         (*********************************************)
         (* parameter 3.4.7 *)
         (*********************************************)
         (
            ParameterName_as8    := 'Output Value 43',
            ParameterType_u8     := 0,
            attr1_u              := 0,
            attr2_u              := 10000,
            attr3_u              := 50,
            UnitCode_au8         := 15,
            Multiplier_s16       := 1,
            Divisor_s16          := 1,
            NumberOfDigits_u16   := 0,
            AccesslevelCode_u8   := 129,
            attr4_u              := 0,
            EEPROMAddress_s      := (Page_u8 := 3, IntIndex_u8 := 158)
         ),

         (*********************************************)
         (* parameter 3.4.8 *)
         (*********************************************)
         (
            ParameterName_as8    := 'Output Value 44',
            ParameterType_u8     := 0,
            attr1_u              := 0,
            attr2_u              := 10000,
            attr3_u              := 50,
            UnitCode_au8         := 15,
            Multiplier_s16       := 1,
            Divisor_s16          := 1,
            NumberOfDigits_u16   := 0,
            AccesslevelCode_u8   := 129,
            attr4_u              := 0,
            EEPROMAddress_s      := (Page_u8 := 3, IntIndex_u8 := 159)
         )

      ),

      (*********************************************)
      (* parameter group 3.5 - up to 8 parameters can be defined here *)
      (*********************************************)
      (
         GroupName_as8   := 'Output Value 45-47',

         Param_as        := 

         (*********************************************)
         (* parameter 3.5.1 *)
         (*********************************************)
         (
            ParameterName_as8    := 'Output Value 45',
            ParameterType_u8     := 0,
            attr1_u              := 0,
            attr2_u              := 10000,
            attr3_u              := 50,
            UnitCode_au8         := 15,
            Multiplier_s16       := 1,
            Divisor_s16          := 1,
            NumberOfDigits_u16   := 0,
            AccesslevelCode_u8   := 129,
            attr4_u              := 0,
            EEPROMAddress_s      := (Page_u8 := 3, IntIndex_u8 := 160)
         ),

         (*********************************************)
         (* parameter 3.5.2 *)
         (*********************************************)
         (
            ParameterName_as8    := 'Output Value 46',
            ParameterType_u8     := 0,
            attr1_u              := 0,
            attr2_u              := 10000,
            attr3_u              := 50,
            UnitCode_au8         := 15,
            Multiplier_s16       := 1,
            Divisor_s16          := 1,
            NumberOfDigits_u16   := 0,
            AccesslevelCode_u8   := 129,
            attr4_u              := 0,
            EEPROMAddress_s      := (Page_u8 := 3, IntIndex_u8 := 161)
         ),

         (*********************************************)
         (* parameter 3.5.3 *)
         (*********************************************)
         (
            ParameterName_as8    := 'Output Value 47',
            ParameterType_u8     := 0,
            attr1_u              := 0,
            attr2_u              := 20000,
            attr3_u              := 50,
            UnitCode_au8         := 15,
            Multiplier_s16       := 1,
            Divisor_s16          := 1,
            NumberOfDigits_u16   := 0,
            AccesslevelCode_u8   := 129,
            attr4_u              := 0,
            EEPROMAddress_s      := (Page_u8 := 3, IntIndex_u8 := 162)
         ),

         (*********************************************)
         (* parameter 3.5.4 *)
         (*********************************************)
         (
         ),

         (*********************************************)
         (* parameter 3.5.5 *)
         (*********************************************)
         (
         ),

         (*********************************************)
         (* parameter 3.5.6 *)
         (*********************************************)
         (
         ),

         (*********************************************)
         (* parameter 3.5.7 *)
         (*********************************************)
         (
         ),

         (*********************************************)
         (* parameter 3.5.8 *)
         (*********************************************)
         (
         )

      ),

      (*********************************************)
      (* parameter group 3.6 - up to 8 parameters can be defined here *)
      (*********************************************)
      (
         GroupName_as8   := 'POH Configuration',

         Param_as        := 

         (*********************************************)
         (* parameter 3.6.1 *)
         (*********************************************)
         (
            ParameterName_as8    := 'POH Debounce',
            ParameterType_u8     := 0,
            attr1_u              := 50,
            attr2_u              := 250,
            attr3_u              := 10,
            UnitCode_au8         := 4,
            Multiplier_s16       := 1,
            Divisor_s16          := 1,
            NumberOfDigits_u16   := 0,
            AccesslevelCode_u8   := 179,
            attr4_u              := 100,
            EEPROMAddress_s      := (Page_u8 := 3, IntIndex_u8 := 168)
         ),

         (*********************************************)
         (* parameter 3.6.2 *)
         (*********************************************)
         (
         ),

         (*********************************************)
         (* parameter 3.6.3 *)
         (*********************************************)
         (
            ParameterName_as8    := 'POH Resistance Min',
            ParameterType_u8     := 0,
            attr1_u              := 0,
            attr2_u              := 3000,
            attr3_u              := 10,
            UnitCode_au8         := 18,
            Multiplier_s16       := 1,
            Divisor_s16          := 1,
            NumberOfDigits_u16   := 0,
            AccesslevelCode_u8   := 179,
            attr4_u              := 2,
            EEPROMAddress_s      := (Page_u8 := 3, IntIndex_u8 := 170)
         ),

         (*********************************************)
         (* parameter 3.6.4 *)
         (*********************************************)
         (
            ParameterName_as8    := 'POH Resistance Max',
            ParameterType_u8     := 0,
            attr1_u              := 0,
            attr2_u              := 3000,
            attr3_u              := 10,
            UnitCode_au8         := 18,
            Multiplier_s16       := 1,
            Divisor_s16          := 1,
            NumberOfDigits_u16   := 0,
            AccesslevelCode_u8   := 179,
            attr4_u              := 52,
            EEPROMAddress_s      := (Page_u8 := 3, IntIndex_u8 := 171)
         ),

         (*********************************************)
         (* parameter 3.6.5 *)
         (*********************************************)
         (
            ParameterName_as8    := 'POH Kp',
            ParameterType_u8     := 0,
            attr1_u              := 0,
            attr2_u              := 2000,
            attr3_u              := 50,
            UnitCode_au8         := 0,
            Multiplier_s16       := 1,
            Divisor_s16          := 1,
            NumberOfDigits_u16   := 0,
            AccesslevelCode_u8   := 179,
            attr4_u              := 250,
            EEPROMAddress_s      := (Page_u8 := 3, IntIndex_u8 := 172)
         ),

         (*********************************************)
         (* parameter 3.6.6 *)
         (*********************************************)
         (
            ParameterName_as8    := 'POH Ki',
            ParameterType_u8     := 0,
            attr1_u              := 0,
            attr2_u              := 500,
            attr3_u              := 50,
            UnitCode_au8         := 0,
            Multiplier_s16       := 1,
            Divisor_s16          := 1,
            NumberOfDigits_u16   := 0,
            AccesslevelCode_u8   := 179,
            attr4_u              := 250,
            EEPROMAddress_s      := (Page_u8 := 3, IntIndex_u8 := 173)
         ),

         (*********************************************)
         (* parameter 3.6.7 *)
         (*********************************************)
         (
         ),

         (*********************************************)
         (* parameter 3.6.8 *)
         (*********************************************)
         (
         )

      ),

      (*********************************************)
      (* parameter group 3.7 - up to 8 parameters can be defined here *)
      (*********************************************)
      (
         GroupName_as8   := 'POL Configuration',

         Param_as        := 

         (*********************************************)
         (* parameter 3.7.1 *)
         (*********************************************)
         (
            ParameterName_as8    := 'POL Debounce',
            ParameterType_u8     := 0,
            attr1_u              := 50,
            attr2_u              := 250,
            attr3_u              := 10,
            UnitCode_au8         := 4,
            Multiplier_s16       := 1,
            Divisor_s16          := 1,
            NumberOfDigits_u16   := 0,
            AccesslevelCode_u8   := 179,
            attr4_u              := 100,
            EEPROMAddress_s      := (Page_u8 := 3, IntIndex_u8 := 176)
         ),

         (*********************************************)
         (* parameter 3.7.2 *)
         (*********************************************)
         (
         ),

         (*********************************************)
         (* parameter 3.7.3 *)
         (*********************************************)
         (
            ParameterName_as8    := 'POL Resistance Min',
            ParameterType_u8     := 0,
            attr1_u              := 0,
            attr2_u              := 3000,
            attr3_u              := 10,
            UnitCode_au8         := 18,
            Multiplier_s16       := 1,
            Divisor_s16          := 1,
            NumberOfDigits_u16   := 0,
            AccesslevelCode_u8   := 179,
            attr4_u              := 2,
            EEPROMAddress_s      := (Page_u8 := 3, IntIndex_u8 := 178)
         ),

         (*********************************************)
         (* parameter 3.7.4 *)
         (*********************************************)
         (
            ParameterName_as8    := 'POL Resistance Max',
            ParameterType_u8     := 0,
            attr1_u              := 0,
            attr2_u              := 3000,
            attr3_u              := 10,
            UnitCode_au8         := 18,
            Multiplier_s16       := 1,
            Divisor_s16          := 1,
            NumberOfDigits_u16   := 0,
            AccesslevelCode_u8   := 179,
            attr4_u              := 52,
            EEPROMAddress_s      := (Page_u8 := 3, IntIndex_u8 := 179)
         ),

         (*********************************************)
         (* parameter 3.7.5 *)
         (*********************************************)
         (
            ParameterName_as8    := 'POL Kp',
            ParameterType_u8     := 0,
            attr1_u              := 0,
            attr2_u              := 2000,
            attr3_u              := 50,
            UnitCode_au8         := 0,
            Multiplier_s16       := 1,
            Divisor_s16          := 1,
            NumberOfDigits_u16   := 0,
            AccesslevelCode_u8   := 179,
            attr4_u              := 250,
            EEPROMAddress_s      := (Page_u8 := 3, IntIndex_u8 := 180)
         ),

         (*********************************************)
         (* parameter 3.7.6 *)
         (*********************************************)
         (
            ParameterName_as8    := 'POL Ki',
            ParameterType_u8     := 0,
            attr1_u              := 0,
            attr2_u              := 500,
            attr3_u              := 50,
            UnitCode_au8         := 0,
            Multiplier_s16       := 1,
            Divisor_s16          := 1,
            NumberOfDigits_u16   := 0,
            AccesslevelCode_u8   := 179,
            attr4_u              := 250,
            EEPROMAddress_s      := (Page_u8 := 3, IntIndex_u8 := 181)
         ),

         (*********************************************)
         (* parameter 3.7.7 *)
         (*********************************************)
         (
         ),

         (*********************************************)
         (* parameter 3.7.8 *)
         (*********************************************)
         (
         )

      ),

      (*********************************************)
      (* parameter group 3.8 - up to 8 parameters can be defined here *)
      (*********************************************)
      (
         GroupName_as8   := 'DOH Configuration',

         Param_as        := 

         (*********************************************)
         (* parameter 3.8.1 *)
         (*********************************************)
         (
            ParameterName_as8    := 'DOH Debounce',
            ParameterType_u8     := 0,
            attr1_u              := 50,
            attr2_u              := 250,
            attr3_u              := 10,
            UnitCode_au8         := 4,
            Multiplier_s16       := 1,
            Divisor_s16          := 1,
            NumberOfDigits_u16   := 0,
            AccesslevelCode_u8   := 179,
            attr4_u              := 200,
            EEPROMAddress_s      := (Page_u8 := 3, IntIndex_u8 := 184)
         ),

         (*********************************************)
         (* parameter 3.8.2 *)
         (*********************************************)
         (
         ),

         (*********************************************)
         (* parameter 3.8.3 *)
         (*********************************************)
         (
            ParameterName_as8    := 'DOH Resistance Min',
            ParameterType_u8     := 0,
            attr1_u              := 0,
            attr2_u              := 3000,
            attr3_u              := 10,
            UnitCode_au8         := 18,
            Multiplier_s16       := 1,
            Divisor_s16          := 1,
            NumberOfDigits_u16   := 0,
            AccesslevelCode_u8   := 179,
            attr4_u              := 6,
            EEPROMAddress_s      := (Page_u8 := 3, IntIndex_u8 := 186)
         ),

         (*********************************************)
         (* parameter 3.8.4 *)
         (*********************************************)
         (
            ParameterName_as8    := 'DOH Resistance Max',
            ParameterType_u8     := 0,
            attr1_u              := 0,
            attr2_u              := 3000,
            attr3_u              := 10,
            UnitCode_au8         := 18,
            Multiplier_s16       := 1,
            Divisor_s16          := 1,
            NumberOfDigits_u16   := 0,
            AccesslevelCode_u8   := 179,
            attr4_u              := 44,
            EEPROMAddress_s      := (Page_u8 := 3, IntIndex_u8 := 187)
         ),

         (*********************************************)
         (* parameter 3.8.5 *)
         (*********************************************)
         (
         ),

         (*********************************************)
         (* parameter 3.8.6 *)
         (*********************************************)
         (
         ),

         (*********************************************)
         (* parameter 3.8.7 *)
         (*********************************************)
         (
         ),

         (*********************************************)
         (* parameter 3.8.8 *)
         (*********************************************)
         (
         )

      )

   ),

   (*********************************************)
   (* parameter menu 4 - up to 8 groups can be defined here *)
   (*********************************************)
   (
      MenuName_as8        := 'Menu 4',

      ParameterGroup_as   := 

      (*********************************************)
      (* parameter group 4.1 - up to 8 parameters can be defined here *)
      (*********************************************)
      (








      ),

      (*********************************************)
      (* parameter group 4.2 - up to 8 parameters can be defined here *)
      (*********************************************)
      (








      ),

      (*********************************************)
      (* parameter group 4.3 - up to 8 parameters can be defined here *)
      (*********************************************)
      (








      ),

      (*********************************************)
      (* parameter group 4.4 - up to 8 parameters can be defined here *)
      (*********************************************)
      (








      ),

      (*********************************************)
      (* parameter group 4.5 - up to 8 parameters can be defined here *)
      (*********************************************)
      (








      ),

      (*********************************************)
      (* parameter group 4.6 - up to 8 parameters can be defined here *)
      (*********************************************)
      (








      ),

      (*********************************************)
      (* parameter group 4.7 - up to 8 parameters can be defined here *)
      (*********************************************)
      (








      ),

      (*********************************************)
      (* parameter group 4.8 - up to 8 parameters can be defined here *)
      (*********************************************)
      (








      )

   ),

   (*********************************************)
   (* parameter menu 5 - up to 8 groups can be defined here *)
   (*********************************************)
   (
      MenuName_as8        := 'Menu 5',

      ParameterGroup_as   := 

      (*********************************************)
      (* parameter group 5.1 - up to 8 parameters can be defined here *)
      (*********************************************)
      (








      ),

      (*********************************************)
      (* parameter group 5.2 - up to 8 parameters can be defined here *)
      (*********************************************)
      (








      ),

      (*********************************************)
      (* parameter group 5.3 - up to 8 parameters can be defined here *)
      (*********************************************)
      (








      ),

      (*********************************************)
      (* parameter group 5.4 - up to 8 parameters can be defined here *)
      (*********************************************)
      (








      ),

      (*********************************************)
      (* parameter group 5.5 - up to 8 parameters can be defined here *)
      (*********************************************)
      (








      ),

      (*********************************************)
      (* parameter group 5.6 - up to 8 parameters can be defined here *)
      (*********************************************)
      (








      ),

      (*********************************************)
      (* parameter group 5.7 - up to 8 parameters can be defined here *)
      (*********************************************)
      (








      ),

      (*********************************************)
      (* parameter group 5.8 - up to 8 parameters can be defined here *)
      (*********************************************)
      (








      )

   );


(**)
END_VAR
(*********************************************)
(*  DON'T MAKE ANY CHANGES TO THIS PROGRAM!! *)
(*     FILE WAS AUTOMATICALLY GENERATED!!    *)
(*********************************************)

;
END_PROGRAM

(* POU Autocode/ProcData, ST *)
PROGRAM ProcData
(*********************************************)
(*  DON'T MAKE ANY CHANGES TO THIS PROGRAM!! *)
(*     FILE WAS AUTOMATICALLY GENERATED!!    *)
(*********************************************)

VAR
END_VAR
VAR CONSTANT

(**)
(*********************************************)
nrProcMenus_u8          : USINT := 48;

(*********************************************)
(* Process Values Tree *)
(*********************************************)

ProcessVarGroups_as      : ARRAY [1..48] OF ProcessVariableGroup_ts := 

   (*********************************************)
   (* process values group 1 - up to 8 variables can be defined here *)
   (*********************************************)
   (
      GroupName_as8        := 'Group 1',

      ProcessVariable_as   := 

         (*********************************************)
         (* process value 1.1 *)
         (*********************************************)
         (
         ProcessVarName_as8   := 'Param_var',
         ProcVarType_u8       := 0,
         UnitCode_au8         := 1,
         Multiplier_s16       := 1,
         Divisor_s16          := 1,
         attr_u               := 0,
         AccesslevelCode_u8   := 129
         ),
         (*********************************************)
         (* process value 1.2 *)
         (*********************************************)
         (
         ProcessVarName_as8   := 'Param_var',
         ProcVarType_u8       := 0,
         UnitCode_au8         := 1,
         Multiplier_s16       := 1,
         Divisor_s16          := 1,
         attr_u               := 0,
         AccesslevelCode_u8   := 129
         ),
         (*********************************************)
         (* process value 1.3 *)
         (*********************************************)
         (
         ProcessVarName_as8   := 'Param_var',
         ProcVarType_u8       := 0,
         UnitCode_au8         := 1,
         Multiplier_s16       := 1,
         Divisor_s16          := 1,
         attr_u               := 0,
         AccesslevelCode_u8   := 129
         ),
         (*********************************************)
         (* process value 1.4 *)
         (*********************************************)
         (
         ProcessVarName_as8   := 'Param_var',
         ProcVarType_u8       := 0,
         UnitCode_au8         := 1,
         Multiplier_s16       := 1,
         Divisor_s16          := 1,
         attr_u               := 0,
         AccesslevelCode_u8   := 129
         ),
         (*********************************************)
         (* process value 1.5 *)
         (*********************************************)
         (
         ProcessVarName_as8   := 'Param_var',
         ProcVarType_u8       := 0,
         UnitCode_au8         := 0,
         Multiplier_s16       := 1,
         Divisor_s16          := 1,
         attr_u               := 0,
         AccesslevelCode_u8   := 129
         ),
         (*********************************************)
         (* process value 1.6 *)
         (*********************************************)
         (
         ProcessVarName_as8   := 'Param_var',
         ProcVarType_u8       := 0,
         UnitCode_au8         := 0,
         Multiplier_s16       := 1,
         Divisor_s16          := 1,
         attr_u               := 15,
         AccesslevelCode_u8   := 129
         ),
         (*********************************************)
         (* process value 1.7 *)
         (*********************************************)
         (
         ProcessVarName_as8   := 'Param_var',
         ProcVarType_u8       := 0,
         UnitCode_au8         := 0,
         Multiplier_s16       := 1,
         Divisor_s16          := 1,
         attr_u               := 8,
         AccesslevelCode_u8   := 129
         ),
         (*********************************************)
         (* process value 1.8 *)
         (*********************************************)
         (
         ProcessVarName_as8   := 'Param_var',
         ProcVarType_u8       := 0,
         UnitCode_au8         := 0,
         Multiplier_s16       := 1,
         Divisor_s16          := 1,
         attr_u               := 1000,
         AccesslevelCode_u8   := 129
         )
   ),

   (*********************************************)
   (* process values group 2 - up to 8 variables can be defined here *)
   (*********************************************)
   (
      GroupName_as8        := 'Group 2',

      ProcessVariable_as   := 

         (*********************************************)
         (* process value 2.1 *)
         (*********************************************)
         (
         ProcessVarName_as8   := 'Param_var',
         ProcVarType_u8       := 0,
         UnitCode_au8         := 1,
         Multiplier_s16       := 1,
         Divisor_s16          := 1,
         attr_u               := 0,
         AccesslevelCode_u8   := 129
         ),
         (*********************************************)
         (* process value 2.2 *)
         (*********************************************)
         (
         ProcessVarName_as8   := 'Param_var',
         ProcVarType_u8       := 0,
         UnitCode_au8         := 1,
         Multiplier_s16       := 1,
         Divisor_s16          := 1,
         attr_u               := 0,
         AccesslevelCode_u8   := 129
         ),
         (*********************************************)
         (* process value 2.3 *)
         (*********************************************)
         (
         ProcessVarName_as8   := 'Param_var',
         ProcVarType_u8       := 0,
         UnitCode_au8         := 1,
         Multiplier_s16       := 1,
         Divisor_s16          := 1,
         attr_u               := 0,
         AccesslevelCode_u8   := 129
         ),
         (*********************************************)
         (* process value 2.4 *)
         (*********************************************)
         (
         ProcessVarName_as8   := 'Param_var',
         ProcVarType_u8       := 0,
         UnitCode_au8         := 1,
         Multiplier_s16       := 1,
         Divisor_s16          := 1,
         attr_u               := 0,
         AccesslevelCode_u8   := 129
         ),
         (*********************************************)
         (* process value 2.5 *)
         (*********************************************)
         (
         ProcessVarName_as8   := 'Param_var',
         ProcVarType_u8       := 0,
         UnitCode_au8         := 1,
         Multiplier_s16       := 1,
         Divisor_s16          := 1,
         attr_u               := 0,
         AccesslevelCode_u8   := 129
         ),
         (*********************************************)
         (* process value 2.6 *)
         (*********************************************)
         (
         ProcessVarName_as8   := 'Param_var',
         ProcVarType_u8       := 0,
         UnitCode_au8         := 1,
         Multiplier_s16       := 1,
         Divisor_s16          := 1,
         attr_u               := 0,
         AccesslevelCode_u8   := 129
         ),
         (*********************************************)
         (* process value 2.7 *)
         (*********************************************)
         (
         ProcessVarName_as8   := 'Param_var',
         ProcVarType_u8       := 0,
         UnitCode_au8         := 1,
         Multiplier_s16       := 1,
         Divisor_s16          := 1,
         attr_u               := 0,
         AccesslevelCode_u8   := 129
         ),
         (*********************************************)
         (* process value 2.8 *)
         (*********************************************)
         (
         ProcessVarName_as8   := 'Param_var',
         ProcVarType_u8       := 0,
         UnitCode_au8         := 1,
         Multiplier_s16       := 1,
         Divisor_s16          := 1,
         attr_u               := 0,
         AccesslevelCode_u8   := 129
         )
   ),

   (*********************************************)
   (* process values group 3 - up to 8 variables can be defined here *)
   (*********************************************)
   (
      GroupName_as8        := 'Group 3',

      ProcessVariable_as   := 

         (*********************************************)
         (* process value 3.1 *)
         (*********************************************)
         (
         ProcessVarName_as8   := 'Param_var',
         ProcVarType_u8       := 0,
         UnitCode_au8         := 1,
         Multiplier_s16       := 1,
         Divisor_s16          := 1,
         attr_u               := 0,
         AccesslevelCode_u8   := 129
         ),
         (*********************************************)
         (* process value 3.2 *)
         (*********************************************)
         (
         ProcessVarName_as8   := 'Param_var',
         ProcVarType_u8       := 0,
         UnitCode_au8         := 1,
         Multiplier_s16       := 1,
         Divisor_s16          := 1,
         attr_u               := 0,
         AccesslevelCode_u8   := 129
         ),
         (*********************************************)
         (* process value 3.3 *)
         (*********************************************)
         (
         ProcessVarName_as8   := 'Param_var',
         ProcVarType_u8       := 0,
         UnitCode_au8         := 1,
         Multiplier_s16       := 1,
         Divisor_s16          := 1,
         attr_u               := 0,
         AccesslevelCode_u8   := 129
         ),
         (*********************************************)
         (* process value 3.4 *)
         (*********************************************)
         (
         ProcessVarName_as8   := 'Param_var',
         ProcVarType_u8       := 0,
         UnitCode_au8         := 1,
         Multiplier_s16       := 1,
         Divisor_s16          := 1,
         attr_u               := 0,
         AccesslevelCode_u8   := 129
         ),
         (*********************************************)
         (* process value 3.5 *)
         (*********************************************)
         (
         ProcessVarName_as8   := 'Param_var',
         ProcVarType_u8       := 0,
         UnitCode_au8         := 1,
         Multiplier_s16       := 1,
         Divisor_s16          := 1,
         attr_u               := 0,
         AccesslevelCode_u8   := 129
         ),
         (*********************************************)
         (* process value 3.6 *)
         (*********************************************)
         (
         ProcessVarName_as8   := 'Param_var',
         ProcVarType_u8       := 0,
         UnitCode_au8         := 1,
         Multiplier_s16       := 1,
         Divisor_s16          := 1,
         attr_u               := 0,
         AccesslevelCode_u8   := 129
         ),
         (*********************************************)
         (* process value 3.7 *)
         (*********************************************)
         (
         ProcessVarName_as8   := 'Param_var',
         ProcVarType_u8       := 0,
         UnitCode_au8         := 1,
         Multiplier_s16       := 1,
         Divisor_s16          := 1,
         attr_u               := 0,
         AccesslevelCode_u8   := 129
         ),
         (*********************************************)
         (* process value 3.8 *)
         (*********************************************)
         (
         ProcessVarName_as8   := 'Param_var',
         ProcVarType_u8       := 0,
         UnitCode_au8         := 1,
         Multiplier_s16       := 1,
         Divisor_s16          := 1,
         attr_u               := 0,
         AccesslevelCode_u8   := 129
         )
   ),

   (*********************************************)
   (* process values group 4 - up to 8 variables can be defined here *)
   (*********************************************)
   (
      GroupName_as8        := 'Group 4',

      ProcessVariable_as   := 

         (*********************************************)
         (* process value 4.1 *)
         (*********************************************)
         (
         ProcessVarName_as8   := 'Param_var',
         ProcVarType_u8       := 0,
         UnitCode_au8         := 1,
         Multiplier_s16       := 1,
         Divisor_s16          := 1,
         attr_u               := 0,
         AccesslevelCode_u8   := 129
         ),
         (*********************************************)
         (* process value 4.2 *)
         (*********************************************)
         (
         ProcessVarName_as8   := 'Param_var',
         ProcVarType_u8       := 0,
         UnitCode_au8         := 1,
         Multiplier_s16       := 1,
         Divisor_s16          := 1,
         attr_u               := 0,
         AccesslevelCode_u8   := 129
         ),
         (*********************************************)
         (* process value 4.3 *)
         (*********************************************)
         (
         ProcessVarName_as8   := 'Param_var',
         ProcVarType_u8       := 0,
         UnitCode_au8         := 1,
         Multiplier_s16       := 1,
         Divisor_s16          := 1,
         attr_u               := 0,
         AccesslevelCode_u8   := 129
         ),
         (*********************************************)
         (* process value 4.4 *)
         (*********************************************)
         (
         ProcessVarName_as8   := 'Param_var',
         ProcVarType_u8       := 0,
         UnitCode_au8         := 1,
         Multiplier_s16       := 1,
         Divisor_s16          := 1,
         attr_u               := 0,
         AccesslevelCode_u8   := 129
         ),
         (*********************************************)
         (* process value 4.5 *)
         (*********************************************)
         (
         ProcessVarName_as8   := 'Param_var',
         ProcVarType_u8       := 0,
         UnitCode_au8         := 1,
         Multiplier_s16       := 1,
         Divisor_s16          := 1,
         attr_u               := 0,
         AccesslevelCode_u8   := 129
         ),
         (*********************************************)
         (* process value 4.6 *)
         (*********************************************)
         (
         ProcessVarName_as8   := 'Param_var',
         ProcVarType_u8       := 0,
         UnitCode_au8         := 1,
         Multiplier_s16       := 1,
         Divisor_s16          := 1,
         attr_u               := 0,
         AccesslevelCode_u8   := 129
         ),
         (*********************************************)
         (* process value 4.7 *)
         (*********************************************)
         (
         ProcessVarName_as8   := 'Param_var',
         ProcVarType_u8       := 0,
         UnitCode_au8         := 1,
         Multiplier_s16       := 1,
         Divisor_s16          := 1,
         attr_u               := 0,
         AccesslevelCode_u8   := 129
         ),
         (*********************************************)
         (* process value 4.8 *)
         (*********************************************)
         (
         )
   ),

   (*********************************************)
   (* process values group 5 - up to 8 variables can be defined here *)
   (*********************************************)
   (
      GroupName_as8        := 'Group 5',

      ProcessVariable_as   := 

         (*********************************************)
         (* process value 5.1 *)
         (*********************************************)
         (
         ProcessVarName_as8   := 'Param_var',
         ProcVarType_u8       := 0,
         UnitCode_au8         := 1,
         Multiplier_s16       := 1,
         Divisor_s16          := 1,
         attr_u               := 0,
         AccesslevelCode_u8   := 129
         ),
         (*********************************************)
         (* process value 5.2 *)
         (*********************************************)
         (
         ProcessVarName_as8   := 'Param_var',
         ProcVarType_u8       := 0,
         UnitCode_au8         := 1,
         Multiplier_s16       := 1,
         Divisor_s16          := 1,
         attr_u               := 0,
         AccesslevelCode_u8   := 129
         ),
         (*********************************************)
         (* process value 5.3 *)
         (*********************************************)
         (
         ProcessVarName_as8   := 'Param_var',
         ProcVarType_u8       := 0,
         UnitCode_au8         := 1,
         Multiplier_s16       := 1,
         Divisor_s16          := 1,
         attr_u               := 0,
         AccesslevelCode_u8   := 129
         ),
         (*********************************************)
         (* process value 5.4 *)
         (*********************************************)
         (
         ProcessVarName_as8   := 'Param_var',
         ProcVarType_u8       := 0,
         UnitCode_au8         := 1,
         Multiplier_s16       := 1,
         Divisor_s16          := 1,
         attr_u               := 0,
         AccesslevelCode_u8   := 129
         ),
         (*********************************************)
         (* process value 5.5 *)
         (*********************************************)
         (
         ProcessVarName_as8   := 'Param_var',
         ProcVarType_u8       := 0,
         UnitCode_au8         := 1,
         Multiplier_s16       := 1,
         Divisor_s16          := 1,
         attr_u               := 0,
         AccesslevelCode_u8   := 129
         ),
         (*********************************************)
         (* process value 5.6 *)
         (*********************************************)
         (
         ProcessVarName_as8   := 'Param_var',
         ProcVarType_u8       := 0,
         UnitCode_au8         := 1,
         Multiplier_s16       := 1,
         Divisor_s16          := 1,
         attr_u               := 0,
         AccesslevelCode_u8   := 129
         ),
         (*********************************************)
         (* process value 5.7 *)
         (*********************************************)
         (
         ),
         (*********************************************)
         (* process value 5.8 *)
         (*********************************************)
         (
         )
   ),

   (*********************************************)
   (* process values group 6 - up to 8 variables can be defined here *)
   (*********************************************)
   (


   ),

   (*********************************************)
   (* process values group 7 - up to 8 variables can be defined here *)
   (*********************************************)
   (


   ),

   (*********************************************)
   (* process values group 8 - up to 8 variables can be defined here *)
   (*********************************************)
   (


   ),

   (*********************************************)
   (* process values group 9 - up to 8 variables can be defined here *)
   (*********************************************)
   (


   ),

   (*********************************************)
   (* process values group 10 - up to 8 variables can be defined here *)
   (*********************************************)
   (


   ),

   (*********************************************)
   (* process values group 11 - up to 8 variables can be defined here *)
   (*********************************************)
   (


   ),

   (*********************************************)
   (* process values group 12 - up to 8 variables can be defined here *)
   (*********************************************)
   (


   ),

   (*********************************************)
   (* process values group 13 - up to 8 variables can be defined here *)
   (*********************************************)
   (


   ),

   (*********************************************)
   (* process values group 14 - up to 8 variables can be defined here *)
   (*********************************************)
   (


   ),

   (*********************************************)
   (* process values group 15 - up to 8 variables can be defined here *)
   (*********************************************)
   (


   ),

   (*********************************************)
   (* process values group 16 - up to 8 variables can be defined here *)
   (*********************************************)
   (


   ),

   (*********************************************)
   (* process values group 17 - up to 8 variables can be defined here *)
   (*********************************************)
   (


   ),

   (*********************************************)
   (* process values group 18 - up to 8 variables can be defined here *)
   (*********************************************)
   (


   ),

   (*********************************************)
   (* process values group 19 - up to 8 variables can be defined here *)
   (*********************************************)
   (


   ),

   (*********************************************)
   (* process values group 20 - up to 8 variables can be defined here *)
   (*********************************************)
   (


   ),

   (*********************************************)
   (* process values group 21 - up to 8 variables can be defined here *)
   (*********************************************)
   (


   ),

   (*********************************************)
   (* process values group 22 - up to 8 variables can be defined here *)
   (*********************************************)
   (


   ),

   (*********************************************)
   (* process values group 23 - up to 8 variables can be defined here *)
   (*********************************************)
   (


   ),

   (*********************************************)
   (* process values group 24 - up to 8 variables can be defined here *)
   (*********************************************)
   (


   ),

   (*********************************************)
   (* process values group 25 - up to 8 variables can be defined here *)
   (*********************************************)
   (


   ),

   (*********************************************)
   (* process values group 26 - up to 8 variables can be defined here *)
   (*********************************************)
   (


   ),

   (*********************************************)
   (* process values group 27 - up to 8 variables can be defined here *)
   (*********************************************)
   (


   ),

   (*********************************************)
   (* process values group 28 - up to 8 variables can be defined here *)
   (*********************************************)
   (


   ),

   (*********************************************)
   (* process values group 29 - up to 8 variables can be defined here *)
   (*********************************************)
   (


   ),

   (*********************************************)
   (* process values group 30 - up to 8 variables can be defined here *)
   (*********************************************)
   (


   ),

   (*********************************************)
   (* process values group 31 - up to 8 variables can be defined here *)
   (*********************************************)
   (


   ),

   (*********************************************)
   (* process values group 32 - up to 8 variables can be defined here *)
   (*********************************************)
   (


   ),

   (*********************************************)
   (* process values group 33 - up to 8 variables can be defined here *)
   (*********************************************)
   (


   ),

   (*********************************************)
   (* process values group 34 - up to 8 variables can be defined here *)
   (*********************************************)
   (


   ),

   (*********************************************)
   (* process values group 35 - up to 8 variables can be defined here *)
   (*********************************************)
   (


   ),

   (*********************************************)
   (* process values group 36 - up to 8 variables can be defined here *)
   (*********************************************)
   (


   ),

   (*********************************************)
   (* process values group 37 - up to 8 variables can be defined here *)
   (*********************************************)
   (


   ),

   (*********************************************)
   (* process values group 38 - up to 8 variables can be defined here *)
   (*********************************************)
   (


   ),

   (*********************************************)
   (* process values group 39 - up to 8 variables can be defined here *)
   (*********************************************)
   (


   ),

   (*********************************************)
   (* process values group 40 - up to 8 variables can be defined here *)
   (*********************************************)
   (


   ),

   (*********************************************)
   (* process values group 41 - up to 8 variables can be defined here *)
   (*********************************************)
   (


   ),

   (*********************************************)
   (* process values group 42 - up to 8 variables can be defined here *)
   (*********************************************)
   (


   ),

   (*********************************************)
   (* process values group 43 - up to 8 variables can be defined here *)
   (*********************************************)
   (


   ),

   (*********************************************)
   (* process values group 44 - up to 8 variables can be defined here *)
   (*********************************************)
   (


   ),

   (*********************************************)
   (* process values group 45 - up to 8 variables can be defined here *)
   (*********************************************)
   (


   ),

   (*********************************************)
   (* process values group 46 - up to 8 variables can be defined here *)
   (*********************************************)
   (


   ),

   (*********************************************)
   (* process values group 47 - up to 8 variables can be defined here *)
   (*********************************************)
   (


   ),

   (*********************************************)
   (* process values group 48 - up to 8 variables can be defined here *)
   (*********************************************)
   (


   );


(**)
END_VAR
(*********************************************)
(*  DON'T MAKE ANY CHANGES TO THIS PROGRAM!! *)
(*     FILE WAS AUTOMATICALLY GENERATED!!    *)
(*********************************************)

;
END_PROGRAM

(* POU Autocode/UnitCodes, ST *)
PROGRAM UnitCodes
(*********************************************)
(*  DON'T MAKE ANY CHANGES TO THIS PROGRAM!! *)
(*     FILE WAS AUTOMATICALLY GENERATED!!    *)
(*********************************************)

VAR
END_VAR
VAR CONSTANT

(**)
(*********************************************)
nrUnitCodes_u8      : USINT := 18;

(*********************************************)
(* Unit Codes Array *)

UnitCodes_cau8      : ARRAY [1..18] OF STRING(8) := 
   '%',
   'rpm',
   'hrs',
   'ms',
   'ccm',
   'mA',
   'bar',
   'mbar',
   'Deg C',
   'min',
   's',
   'km/h',
   'Nm',
   'deg °',
   '% / mA',
   '% / mV',
   'uA / mV',
   'Ohm';


(**)
END_VAR
(*********************************************)
(*  DON'T MAKE ANY CHANGES TO THIS PROGRAM!! *)
(*     FILE WAS AUTOMATICALLY GENERATED!!    *)
(*********************************************)

;
END_PROGRAM

(* POU Autocode/Lists, ST *)
PROGRAM Lists
(*********************************************)
(*  DON'T MAKE ANY CHANGES TO THIS PROGRAM!! *)
(*     FILE WAS AUTOMATICALLY GENERATED!!    *)
(*********************************************)

VAR
END_VAR
VAR CONSTANT

(**)
(*********************************************)
nrLists_u8      : USINT := 4;

(*********************************************)
(* Lists Tree*)

ParaLists_as      : ARRAY [1..4] OF ARRAY[1..10] OF STRING(32) := 
      'Not Active',
      'Active',
      '',
      '',
      '',
      '',
      '',
      '',
      '',
      '',
      'PWM',
      'PWM Current control',
      '',
      '',
      '',
      '',
      '',
      '',
      '',
      '',
      'PWM',
      'AOV',
      '',
      '',
      '',
      '',
      '',
      '',
      '',
      '',
      'AOC',
      'AOV',
      '',
      '',
      '',
      '',
      '',
      '',
      '',
      ''
;

(**)
END_VAR
(*********************************************)
(*  DON'T MAKE ANY CHANGES TO THIS PROGRAM!! *)
(*     FILE WAS AUTOMATICALLY GENERATED!!    *)
(*********************************************)

;
END_PROGRAM
